PROGRAM Drive_Communication
VAR
	Rotor_Active_Torque AT %I*: INT;	//Rotor Torque as percentage of Rated Motor Torque
	Rotor_Active_Torque_REAL : REAL;
	Rotor_Displayed_Torque :REAL;

	//Feedroll Drive
	Feedroll_Drive_Message AT %I* : USINT;		//Drive Faults
	Feedroll_Drive_Status AT %I* : UINT;
	Feedroll_Drive_Running AT %I* : BOOL;

	
	
	//Rotor Drive
	Rotor_Drive_Message AT %I* : USINT;		//Drive Faults
	Rotor_Drive_Status AT %I* : UINT;
	Rotor_Drive_Running AT %I* : BOOL;


	
	
END_VAR


/////////////////////////Rotor Torque Display Scaling
IF Rotor_Active_Torque < 0 THEN
	Rotor_Active_Torque := Rotor_Active_Torque * -1;
END_IF
Rotor_Active_Torque_REAL := INT_TO_REAL(Rotor_Active_Torque);
Rotor_Displayed_Torque := Rotor_Active_Torque_REAL / 10;



////////////////////////////////////Combined Running Status
IF Feedroll_Drive_Running AND Rotor_Drive_Running THEN
	GVL.Pelletizer_Running := TRUE;
ELSE
	GVL.Pelletizer_Running := FALSE;
END_IF

END_PROGRAM

(* stored: Version 1.1.0.1, ProductVersion 3.1.4024.12
   POU Drive_Communication: Id {f11b8a3c-ca1f-4ae0-8a80-7f86046c4783}, SpecialFunc None *)
